// TIA Portal V19 export
DATA_BLOCK "Mixer_Block_DB"   // DB5
// stored: InstanceOfName Mixer_Block, InstanceOfType FB
"Mixer_Block"
BEGIN
END_DATA_BLOCK
